Universal Robots PolyScope program: ScrewLineProgram.urp

Program ScrewLineProgram (installation=default directory=/home/ur/ursim-current/programs createdIn=5.25.2 lastSavedIn=5.25.2 robotSerialNumber=20195599999)
Calibrated DH parameters: a=[0, -0.425, -0.3922, 0, 0, 0]; d=[0.1625, 0, 0, 0.1333, 0.0997, 0.0996]; alpha=[1.570796, 0, 0, 1.570796, -1.570796, 0]; deltaTheta=[0, 0, 0, 0, 0, 0]
InitVariablesNode variables(variable(name=Heartbeat, expression=0), variable(name=SetPosition, expression=0), variable(name=TargPose, expression=ScrewLine), variable(name=TargPosition, expression=0))
Robot Program (runOnlyOnce=false)
  Set DigitalOutput pin=digital_out[1]; digitalValue=0
  Wait Condition expression=read_port_bit(16)  and read_port_bit(18)
  SetPosition := read_port_register(128)
  TargPosition := SetPosition/10000.0
  TargPose := pose_trans(ScrewLine, p[0,TargPosition, 0, 0, 0, 0])
  MoveL speed 250 mm/s, acceleration 1200 mm/s^2 (useActiveTCP=true optimoveEnabled=false optiMoveSpeed=0.3 optiMoveAcceleration=0.09) feature=Base
    Waypoint Variable (Variable): variable=TargPose
  Set DigitalOutput pin=digital_out[1]; digitalValue=1
  Wait Condition expression=read_port_bit(16)≟ False
  Set DigitalOutput pin=digital_out[1]; digitalValue=0
Thread Thread_1 (runOnlyOnce=false)
  Script: write_port_register(129, read_port_register(128))
  Heartbeat := Heartbeat+1
  If Heartbeat>1000
    Heartbeat := 0
  Script: write_port_register(130, Heartbeat)
  Wait Sleep waitTime=0.05
